{attribute 'reflection'} 
{attribute 'no_explicit_call' := 'do not call this POU directly'} 
FUNCTION_BLOCK FB_EC_MASTER IMPLEMENTS I_Master
VAR_INPUT
END_VAR
VAR_OUTPUT
END_VAR
VAR
	
	{attribute 'instance-path'} 
    {attribute 'noinit'} 
	strInstancePath: STRING;
	strFullObjectPath: STRING;
	stEvent: ST_EVENT;
	bAck: BOOL;
	
	uiDevState AT %I*: 	UINT;
	uiLastDevState: 	UINT;
	
	itfLogEvents: 		I_HANDLE_EVENTS;
	fbEventState: 		FB_CREATE_EVENT(itfLogEvents:= itfLogEvents, itfID:=THIS^);
	bAnyEvent:			BOOL;
END_VAR

METHOD FB_init : BOOL
VAR_INPUT
	bInitRetains : BOOL; // if TRUE, the retain variables are initialized (warm start / cold start)
	bInCopyCode : BOOL;  // if TRUE, the instance afterwards gets moved into the copy code (online change)
	itfLogEvents: 		I_HANDLE_EVENTS;
END_VAR
this^.itfLogEvents:=itfLogEvents;
END_METHOD


(*=== Method: M_Run  ============================================

 @brief: Here is the global code (Timer, Event, Flange,...)*)
METHOD M_Run
VAR
strTemp: STRING;	
END_VAR
//Get own Name
THIS^.strFullObjectPath:= F_RET_TXTLIST_ENTRY(strPortNr:='851', strID:=THIS^.strInstancePath, strTxtLstName:='TXT_LIST_OBJECTS');
bAnyEvent:=FALSE;

//0x0001 = Link error
strTemp:= Tc2_Standard.CONCAT(THIS^.strFullObjectPath, ' -> ');
strTemp:=Tc2_Standard.CONCAT(strTemp, 'Link error');
IF THIS^.uiDevState = 16#0001 THEN
	THIS^.fbEventState.M_Log(strTemp,enum_event_type.Ye4_Stateinfo,THIS^.itfLogEvents);
	bAnyEvent:=TRUE;
END_IF
//0x0002 = I/O locked after link error (I/O reset required)
strTemp:= Tc2_Standard.CONCAT(THIS^.strFullObjectPath, ' -> ');
strTemp:=Tc2_Standard.CONCAT(strTemp, 'I/O locked after link error (I/O reset required)');
IF THIS^.uiDevState = 16#0002 THEN
	THIS^.fbEventState.M_Log(strTemp,enum_event_type.Ye4_Stateinfo,THIS^.itfLogEvents);
	bAnyEvent:=TRUE;
END_IF
//0x0004 = Link error (redundancy adapter)
strTemp:= Tc2_Standard.CONCAT(THIS^.strFullObjectPath, ' -> ');
strTemp:=Tc2_Standard.CONCAT(strTemp, 'Link error (redundancy adapter)');
IF THIS^.uiDevState = 16#0004 THEN
	THIS^.fbEventState.M_Log(strTemp,enum_event_type.Ye4_Stateinfo,THIS^.itfLogEvents);
	bAnyEvent:=TRUE;
END_IF
//0x0008 = Missing one frame (redundancy mode)
strTemp:= Tc2_Standard.CONCAT(THIS^.strFullObjectPath, ' -> ');
strTemp:=Tc2_Standard.CONCAT(strTemp, 'Missing one frame (redundancy mode)');
IF THIS^.uiDevState = 16#0008 THEN
	THIS^.fbEventState.M_Log(strTemp,enum_event_type.Ye4_Stateinfo,THIS^.itfLogEvents);
	bAnyEvent:=TRUE;
END_IF
//0x0010 = Out of send resources (I/O reset required)
strTemp:= Tc2_Standard.CONCAT(THIS^.strFullObjectPath, ' -> ');
strTemp:=Tc2_Standard.CONCAT(strTemp, 'Out of send resources (I/O reset required)');
IF THIS^.uiDevState = 16#0010 THEN
	THIS^.fbEventState.M_Log(strTemp,enum_event_type.Ye4_Stateinfo,THIS^.itfLogEvents);
	bAnyEvent:=TRUE;
END_IF
//0x0020 = Watchdog triggered
strTemp:= Tc2_Standard.CONCAT(THIS^.strFullObjectPath, ' -> ');
strTemp:=Tc2_Standard.CONCAT(strTemp, 'Watchdog triggered');
IF THIS^.uiDevState = 16#0020 THEN
	THIS^.fbEventState.M_Log(strTemp,enum_event_type.Ye4_Stateinfo,THIS^.itfLogEvents);
	bAnyEvent:=TRUE;
END_IF
//0x0040 = Ethernet driver (miniport) not found
strTemp:= Tc2_Standard.CONCAT(THIS^.strFullObjectPath, ' -> ');
strTemp:=Tc2_Standard.CONCAT(strTemp, 'Ethernet driver (miniport) not found');
IF THIS^.uiDevState = 16#0040 THEN
	THIS^.fbEventState.M_Log(strTemp,enum_event_type.Ye4_Stateinfo,THIS^.itfLogEvents);
	bAnyEvent:=TRUE;
END_IF
//0x0080 = I/O reset active
strTemp:= Tc2_Standard.CONCAT(THIS^.strFullObjectPath, ' -> ');
strTemp:=Tc2_Standard.CONCAT(strTemp, 'I/O reset active');
IF THIS^.uiDevState = 16#0080 THEN
	THIS^.fbEventState.M_Log(strTemp,enum_event_type.Ye4_Stateinfo,THIS^.itfLogEvents);
	bAnyEvent:=TRUE;
END_IF
//0x0100 = At least one device in 'INIT' state
strTemp:= Tc2_Standard.CONCAT(THIS^.strFullObjectPath, ' -> ');
strTemp:=Tc2_Standard.CONCAT(strTemp, 'At least one device in "INIT" state');
IF THIS^.uiDevState = 16#0100 THEN
	THIS^.fbEventState.M_Log(strTemp,enum_event_type.Ye4_Stateinfo,THIS^.itfLogEvents);
	bAnyEvent:=TRUE;
END_IF
//0x0200 = At least one device in 'PRE-OP' state
strTemp:= Tc2_Standard.CONCAT(THIS^.strFullObjectPath, ' -> ');
strTemp:=Tc2_Standard.CONCAT(strTemp, 'At least one device in "PRE-OP" state');
IF THIS^.uiDevState = 16#0200 THEN
	THIS^.fbEventState.M_Log(strTemp,enum_event_type.Ye4_Stateinfo,THIS^.itfLogEvents);
	bAnyEvent:=TRUE;
END_IF
//0x0400 = At least one device in 'SAFE-OP' state
strTemp:= Tc2_Standard.CONCAT(THIS^.strFullObjectPath, ' -> ');
strTemp:=Tc2_Standard.CONCAT(strTemp, 'At least one device in "SAFE-OP" state');
IF THIS^.uiDevState = 16#0400 THEN
	THIS^.fbEventState.M_Log(strTemp,enum_event_type.Ye4_Stateinfo,THIS^.itfLogEvents);
	bAnyEvent:=TRUE;
END_IF
//0x0800 = At least one device indicates an error state
strTemp:= Tc2_Standard.CONCAT(THIS^.strFullObjectPath, ' -> ');
strTemp:=Tc2_Standard.CONCAT(strTemp, 'At least one device indicates an error stat');
IF THIS^.uiDevState = 16#0800 THEN
	THIS^.fbEventState.M_Log(strTemp,enum_event_type.Ye4_Stateinfo,THIS^.itfLogEvents);
	bAnyEvent:=TRUE;
END_IF
//0x1000 = DC not in sync
strTemp:= Tc2_Standard.CONCAT(THIS^.strFullObjectPath, ' -> ');
strTemp:=Tc2_Standard.CONCAT(strTemp, 'DC not in sync');
IF THIS^.uiDevState = 16#1000 THEN
	THIS^.fbEventState.M_Log(strTemp,enum_event_type.Ye4_Stateinfo,THIS^.itfLogEvents);
	bAnyEvent:=TRUE;
END_IF




IF THIS^.uiDevState <= 0 
OR THIS^.bAck 
OR NOT bAnyEvent 
OR THIS^.uiLastDevState <>THIS^.uiDevState 
THEN	
	THIS^.fbEventState.M_Log('',enum_event_type.Gn0_None,THIS^.itfLogEvents);
	THIS^.fbEventState.M_Quit();
END_IF
THIS^.uiLastDevState:=THIS^.uiDevState;
END_METHOD

(*=== Property: P_Event  ============================================

 @param [set]: 	Set the Structure "ST_EVENT" from another Object
 @param [get]: 	Return the Structure "ST_EVENT", it contains the actual 
					event of the Object *)
PROPERTY P_Event : GenLib.ST_EVENT
GET
P_Event:= THIS^.stEvent;
END_GET
SET
THIS^.stEvent:=P_Event;
END_SET
END_PROPERTY

(*=== Property: P_FullObjectPath  ============================================

 @param [set]: 	Set the Object Path (Clear String of Object)
 @param [get]: 	Return the Objectpath *)
PROPERTY P_FullObjectPath : STRING
GET
P_FullObjectPath:= THIS^.strFullObjectPath;
END_GET
SET
THIS^.strFullObjectPath:=P_FullObjectPath;
END_SET
END_PROPERTY

(*=== Property: P_Global_Ack  ============================================

 @param [set]: 	Set the Bit for Ack from another Object
 @param [get]: 	Return the state of Ack Bit*)
PROPERTY P_Global_Ack : BOOL
GET
P_Global_Ack:= bAck;
END_GET
SET
bAck:=P_Global_Ack;
END_SET
END_PROPERTY

(*=== Property: P_GlobalID  ============================================

 @param [set]: 	-
 @param [get]: 	Return the string of instance path*)
PROPERTY P_GlobalID : STRING
GET
P_GlobalID:= THIS^.strInstancePath;
END_GET
END_PROPERTY

PROPERTY P_STATE : INT
GET
P_STATE:=UINT_TO_INT(this^.uiDevState);
END_GET
END_PROPERTY

END_FUNCTION_BLOCK

(* stored: Version 1.1.0.1, ProductVersion 3.1.4024.12
   POU FB_EC_MASTER: Id {d6c65fb4-b47e-42b8-ab27-727a51a8839d}, SpecialFunc None
   Method FB_init: Id {e4092c80-6abe-4eed-b559-be5dfe723d25}
   Method M_Run: Id {04314c02-bc79-4d30-bf79-14244a1f5034}
   Property P_Event: Id {618a0041-c8ba-48d8-ab57-77e3756dfda3}
   Get Get: Id {09d7528a-331a-481e-9382-679728d111b1}
   Set Set: Id {4f12f026-b7d8-42b2-9470-8385fc800f0a}
   Property P_FullObjectPath: Id {9246022e-aa34-4db6-99c2-791948feebe9}
   Get Get: Id {6326d28a-8327-4943-93db-d397a80ec55f}
   Set Set: Id {9c1cb438-122b-4702-a3e1-0279a3f306b2}
   Property P_Global_Ack: Id {68141b4e-2099-42bc-9df5-87cd8cf11a75}
   Get Get: Id {7b90b0bb-df90-48d3-9736-4fe573172797}
   Set Set: Id {e37027f3-2910-4c67-a4e4-0975abba8433}
   Property P_GlobalID: Id {cdf44a49-8a1f-4c75-bf55-0d7881e24599}
   Get Get: Id {1368ceed-0543-4886-9bcd-493a9a31e0af}
   Property P_STATE: Id {b8c18c9e-fc22-4423-b5b1-fde46bc54c48}
   Get Get: Id {28e679a9-18de-4834-9547-634651727ae1} *)
